// TIA Portal project "2022.06.10_标准模拟量输出控制变频器" (V17)

(* hardware
DEVICE "S7-1200 station_1"  S7-1200 Station
   slot 0: "Rack_0"  S7-1200 Rack  Rack  V1.0
   slot 1: "PLC_1"  CPU 1212C DC/DC/DC  6ES7 212-1AE40-0XB0  V4.5
   slot 2: "AI 4x13BIT/AQ 2x14BIT_1"  SM 1234 AI4/AQ2  6ES7 234-4HE30-0XB0  V1.0
*)

// ===== PLC "PLC_1"  CPU 1212C DC/DC/DC =====

VAR_GLOBAL   // PLC tag table "默认变量表"
   "所需频率" AT %IW96 : Word;
   "百分比" AT %MD40 : DWord;
   "模拟量输出通道" AT %MD44 : UDInt;
   "所需频率(1)" AT %MD0 : Real;
END_VAR

ORGANIZATION_BLOCK "Main"   // OB1, LAD, ProgramCycle
TITLE = "Main Program Sweep (Cycle)"
{ S7_Optimized_Access := 'TRUE' }
VERSION : 0.1
   VAR_INPUT
      Initial_Call : Bool;   // Initial call of this OB
      Remanence : Bool;   // =True, if remanent data are available
   END_VAR
BEGIN

REGION Network 1
   // 通道0接0-20ma电流信号，通道地址是iw96，对应实际工程中的0-50mpa，将0-27648转换成百分比输出
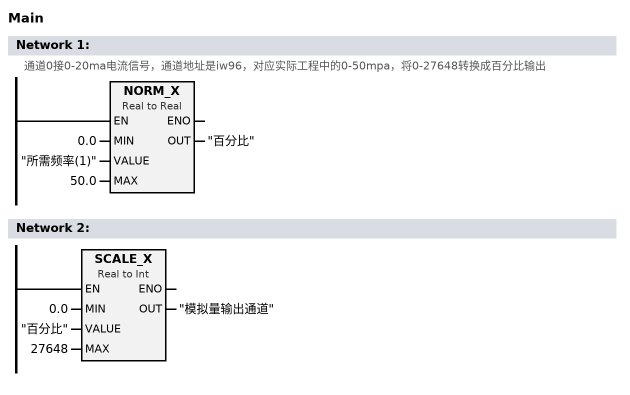
   RUNG wire#powerrail
      { S7_Templates := "[SrcType := Real, DestType := Real]" } Normalize(min := 0.0, value := "所需频率(1)", max := 50.0, out => "百分比")
   END_RUNG
   // the same network as SCL:
   "百分比" := NORM_X(MIN := 0.0, VALUE := "所需频率(1)", MAX := 50.0);
END_REGION

REGION Network 2
   RUNG wire#powerrail
      { S7_Templates := "[SrcType := Real, DestType := Int]" } Scale(min := 0.0, value := "百分比", max := 27648, out => "模拟量输出通道")
   END_RUNG
   // the same network as SCL:
   "模拟量输出通道" := SCALE_X(MIN := 0.0, VALUE := "百分比", MAX := 27648);
END_REGION
END_ORGANIZATION_BLOCK